INTERFACE I_Thermostat

PROPERTY rRequestedTemperature : REAL
GET
END_GET
SET
END_SET
END_PROPERTY

PROPERTY rTemperature : REAL
GET
END_GET
END_PROPERTY

PROPERTY sLocation : STRING
GET
END_GET
END_PROPERTY

PROPERTY sName : String
GET
END_GET
END_PROPERTY

END_INTERFACE

(* stored: Version 1.1.0.1
   Itf I_Thermostat: Id {21e5a810-7393-43f6-8d74-6ffb7812c432}
   Property rRequestedTemperature: Id {3e95d6c7-d820-40ba-9f33-5ade74217fb0}
   Get Get: Id {460a4531-f329-4556-b13a-1d15a832a946}
   Set Set: Id {15c205cb-925e-466e-8817-82e99fa0eb3f}
   Property rTemperature: Id {89f2d91b-b9f3-48bd-8497-b5069f7f3031}
   Get Get: Id {3ed5f81b-28c5-4c49-99ba-dd36ad5fb036}
   Property sLocation: Id {ea5b562b-c68a-4113-ac6d-af3d17be6993}
   Get Get: Id {ff15899d-b8ca-49a7-b60a-112c0f653d1f}
   Property sName: Id {268e05d3-97bd-4a54-bf5c-bf6069140488}
   Get Get: Id {1f848757-a42e-4875-8c1e-a1a81a46c2e4} *)
